Staubli VAL3: RemoteControl.pjx

--- RemoteControl.pjx ---
Parameters version=s8.10.3Cs9_BS2093 stackSize=5000 millimeterUnit=true
Program file=decodeBlend.pgx
Program file=decodeConfig.pgx
Program file=decodeDesc.pgx
Program file=decodeLocation.pgx
Program file=decodePose.pgx
Program file=decodeTool.pgx
Program file=encodeJoint.pgx
Program file=encodePoint.pgx
Program file=init.pgx
Program file=motionReporter.pgx
Program file=motionSupervisor.pgx
Program file=motionWorker.pgx
Program file=movingReporter.pgx
Program file=sendAck.pgx
Program file=sendError.pgx
Program file=sendMoving.pgx
Program file=sendPowerOff.pgx
Program file=sendStatus.pgx
Program file=socketHandler.pgx
Program file=start.pgx
Program file=stop.pgx
Data file=RemoteControl.dtx

--- RemoteControl.dtx ---
num VERSION = 1
sio socket = {link=UdpSocket\RemoteControl}
pointRx BASE_POSITION = {x=50, y=50, z=300, shoulder=sfree, elbow=efree, wrist=wfree, fatherId=world[0]}
jointRx BASE_POSE = {j1=-4.75879959898819E-06, j2=-86.5939224981684, j3=136.317941524159, j4=3.68060849006858E-06, j5=40.2759589805294, j6=-2.91771227743379E-06}
num MAGIC_HEADER = 149
string TASK_NAMES{}
  [MotionWorker] = "motionWorker"
  [MotionReporter] = "motionReporter"
  [MotionSupervisor] = "motionSupervisor"
  [SocketHandler] = "socketHandler"
  [MovingReporter] = "movingReporter"
tool endEffector = {x=660, fatherId=mount[0]}
tool mount = {ry=-90, fatherId=flange[0]}
bool motionQueued
num motionType
num reportInterval
pointRx target = {shoulder=sfree, elbow=efree, wrist=wfree, fatherId=world[0]}
mdesc NOMINAL_CONFIG = {accel=25, decel=25, blend=off}
mdesc SLOW_CONFIG = {accel=25, decel=25, tmax=150, rmax=50, blend=off}
mdesc moveConfig = {blend=off}
jointRx pose
tool selectedTool = {fatherId=flange[0]}
bool reportEnabled
configRx ARM_CONFIG = {shoulder=sfree, elbow=efree, wrist=wfree}
pointRx intermediate = {fatherId=world[0]}

--- start.pgx ---
program start()
begin
  logMsg("RemoteControl - Version " + toString("", VERSION))

  call init()
  enablePower()

  // Move to the initial starting pose
  logMsg("[INIT] Moving dangerously to starting position")
  movej(BASE_POSE, mount, SLOW_CONFIG)
  waitEndMove()

  taskCreate TASK_NAMES["SocketHandler"], 5, socketHandler()
  taskCreate TASK_NAMES["MotionWorker"], 10, motionWorker()
  taskCreate TASK_NAMES["MotionSupervisor"], 20, motionSupervisor()
  taskCreate TASK_NAMES["MovingReporter"], 29, movingReporter()
  taskCreate TASK_NAMES["MotionReporter"], 30, motionReporter()
end

--- decodeBlend.pgx ---
program decodeBlend(mdesc& value, num& buffer[])
  local num decodeBuffer[2]
begin
  if buffer[0] == 0
    value.blend = off
  elseIf buffer[0] == 1
    value.blend = joint
  elseIf buffer[0] == 2
    value.blend = Cartesian
  endIf

  fromBinary(buffer[1], 8, "4.0b", decodeBuffer)

  value.leave = decodeBuffer[0]
  value.reach = decodeBuffer[1]

  logMsg("B: (" + toString("", value.blend) + ", " + toString("", value.leave) + ", " + toString("", value.reach) + ")")
end

--- decodeConfig.pgx ---
program decodeConfig(pointRx& value, num& buffer[])
begin
  if buffer[0] == 0
    value.config.shoulder = sfree
  elseIf buffer[0] == 1
    value.config.shoulder = ssame
  elseIf buffer[0] == 2
    value.config.shoulder = righty
  elseIf buffer[0] == 3
    value.config.shoulder = lefty
  endIf

  if buffer[1] == 0
    value.config.elbow = efree
  elseIf buffer[1] == 1
    value.config.elbow = esame
  elseIf buffer[1] == 2
    value.config.elbow = epositive
  elseIf buffer[1] == 3
    value.config.elbow = enegative
  endIf

  if buffer[2] == 0
    value.config.wrist = wfree
  elseIf buffer[2] == 1
    value.config.wrist = wsame
  elseIf buffer[2] == 2
    value.config.wrist = wpositive
  elseIf buffer[2] == 3
    value.config.wrist = wnegative
  endIf

  logMsg("S: " + toString("", buffer[0]) + "  E: " + toString("", buffer[1]) + "  W: " + toString("", buffer[2]))
end

--- decodeDesc.pgx ---
program decodeDesc(mdesc& value, num& buffer[])
  local num decodeBuffer[3]
begin
  fromBinary(buffer, 8, "4.0b", decodeBuffer)

  value.tvel = decodeBuffer[0]
  value.rvel = decodeBuffer[1]

  fromBinary(buffer[8], 3, "1", decodeBuffer)
  value.accel = decodeBuffer[0]
  value.vel   = decodeBuffer[1]
  value.decel = decodeBuffer[2]

  logMsg("D: (" + toString("3", value.tvel) + ", " + toString("3", value.rvel) + ", " + toString("3", value.accel) + ", " + toString("3", value.vel) + ", " + toString("3", value.decel) + ")")
end

--- decodeLocation.pgx ---
program decodeLocation(point& value, num& buffer[])
  local num decodeBuffer[6]
begin
  fromBinary(buffer, 24, "4.0b", decodeBuffer)

  value.trsf = {decodeBuffer[0], decodeBuffer[1], decodeBuffer[2], decodeBuffer[3], decodeBuffer[4], decodeBuffer[5]}

  logMsg("P: (" + toString("3", value.trsf.x) + ", " + toString("3", value.trsf.y) + ", " + toString("3", value.trsf.z) + ")  R: (" + toString("3", value.trsf.rx) + ", " + toString("3", value.trsf.ry) + ", " + toString("3", value.trsf.rz) + ")")
end

--- decodePose.pgx ---
program decodePose(joint& value, num& buffer[])
  local num decodeBuffer[6]
begin
  fromBinary(buffer, 24, "4.0b", decodeBuffer)

  value = {decodeBuffer[0], decodeBuffer[1], decodeBuffer[2], decodeBuffer[3], decodeBuffer[4], decodeBuffer[5]}

  logMsg("J: (" + toString("3", value.j1) + ", " + toString("3", value.j2) + ", " + toString("3", value.j3) + ", " + toString("3", value.j4) + ", " + toString("3", value.j5) + ", " + toString("3", value.j6) + ")")
end

--- decodeTool.pgx ---
program decodeTool(tool& value, num& buffer[])
  local num decodeBuffer[6]
begin
  fromBinary(buffer, 24, "4.0b", decodeBuffer)

  value.trsf = {decodeBuffer[0], decodeBuffer[1], decodeBuffer[2], decodeBuffer[3], decodeBuffer[4], decodeBuffer[5]}

  logMsg("P: (" + toString("3", value.trsf.x) + ", " + toString("3", value.trsf.y) + ", " + toString("3", value.trsf.z) + ")  R: (" + toString("3", value.trsf.rx) + ", " + toString("3", value.trsf.ry) + ", " + toString("3", value.trsf.rz) + ")")
end

--- encodeJoint.pgx ---
program encodeJoint(joint& value, num& buffer[])
  local num elements[6]
begin
  elements[0] = value.j1
  elements[1] = value.j2
  elements[2] = value.j3
  elements[3] = value.j4
  elements[4] = value.j5
  elements[5] = value.j6

  toBinary(elements, 6, "4.0b", buffer)
end

--- encodePoint.pgx ---
program encodePoint(point& value, num& buffer[])
  local num elements[6]
begin
  elements[0] = value.trsf.x
  elements[1] = value.trsf.y
  elements[2] = value.trsf.z
  elements[3] = value.trsf.rx
  elements[4] = value.trsf.ry
  elements[5] = value.trsf.rz

  toBinary(elements, 6, "4.0b", buffer)
end

--- init.pgx ---
program init()
begin
  moveConfig = NOMINAL_CONFIG
  motionQueued = false
  reportEnabled = false
  reportInterval = 0.1
  selectedTool = endEffector
  target.config = ARM_CONFIG
end

--- motionReporter.pgx ---
program motionReporter()
begin
  while true
    wait(reportEnabled)

    while reportEnabled
      call sendStatus()
      delay(reportInterval)
    endWhile
  endWhile
end

--- motionSupervisor.pgx ---
program motionSupervisor()
  local num buffer[8]
  local num value
begin
  while true
    // Sleep until the task enters a runtime error state
    wait(taskStatus(TASK_NAMES["MotionWorker"]) > 1)

    // Clear any invalid pending trajectories
    resetMotion()

    // Notify any clients of the error
    call sendError(1, taskStatus(TASK_NAMES["MotionWorker"]))

    // Resume the task from the next line
    taskResume(TASK_NAMES["MotionWorker"], 1)
  endWhile
end

--- motionWorker.pgx ---
program motionWorker()
begin

  while true
    wait(motionQueued)
    motionQueued = false

    if motionType == 0
      logMsg("[MOTION] Linear move")
      movel(target, selectedTool, moveConfig)

    elseIf motionType == 1
      logMsg("[MOTION] Direct move")
      movej(target, selectedTool, moveConfig)

    elseIf motionType == 2
      logMsg("[MOTION] Joint move")
      movej(pose, selectedTool, moveConfig)

    elseIf motionType == 3
      logMsg("[MOTION] Circular move")
      movec(intermediate, target, selectedTool, moveConfig)
    endIf

  endWhile
end

--- movingReporter.pgx ---
program movingReporter()
  local bool settled
begin
  settled = false

  while true
    wait(isSettled() != settled)
    settled = !settled

    call sendMoving()
  endWhile
end

--- sendAck.pgx ---
program sendAck(num id)
  local num buffer[3]
begin
  buffer[0] = MAGIC_HEADER
  buffer[1] = 128
  buffer[2] = id
  sioSet(socket, buffer)
end

--- sendComplete.pgx ---
program sendComplete()
  local num buffer[2]
begin
  buffer[0] = MAGIC_HEADER
  buffer[1] = 2
  sioSet(socket, buffer)
end

--- sendError.pgx ---
program sendError(num code, num argument)
  local num buffer[5]
begin
  buffer[0] = MAGIC_HEADER
  buffer[1] = 129
  buffer[2] = code

  toBinary(argument, 1, "2b", buffer[3])

  sioSet(socket, buffer)
end

--- sendMoving.pgx ---
program sendMoving()
  local num buffer[4]
begin
  buffer[0] = MAGIC_HEADER
  buffer[1] = 132
  buffer[2] = sel(isSettled(), 1, 0)
  sioSet(socket, buffer)
end

--- sendPowerOff.pgx ---
program sendPowerOff()
  local num buffer[2]
begin
  buffer[0] = MAGIC_HEADER
  buffer[1] = 130
  sioSet(socket, buffer)
end

--- sendStatus.pgx ---
program sendStatus()
  local num buffer[79]
  local point currentPosition
  local joint currentPose
  local num moveId
begin
  buffer[0] = MAGIC_HEADER
  buffer[1] = 131

  currentPosition = here(endEffector, world)
  call encodePoint(currentPosition, buffer[2])

  currentPose = herej()
  call encodeJoint(currentPose, buffer[26])

  currentPose = getPositionErr()
  call encodeJoint(currentPose, buffer[50])

  buffer[74] = sel(isSettled(), 1, 0)

  moveId = getMoveId()
  toBinary(moveId, 1, "4.0b", buffer[75])

  sioSet(socket, buffer)
end

--- socketHandler.pgx ---
program socketHandler()
  local bool ack
  local num buffer[1024]
  local num bytesRead
  local num payloadSize
begin
  while true
    ack = true
    bytesRead = sioGet(socket, buffer)

    if bytesRead > 0
      logMsg("[SOCKET] UDP packet (" + toString("", bytesRead) + " B)")
    endIf

    if bytesRead >= 3
      payloadSize = bytesRead - 3
    endIf

    if bytesRead < 3
      logMsg("[SOCKET] Too few bytes read, misconfigured socket timeout?", 2)
      ack = false

    elseIf buffer[0] != MAGIC_HEADER
      logMsg("[SOCKET] Missing magic header", 3)
      ack = false

    elseIf buffer[2] == 0 and payloadSize == 0
      logMsg("[SOCKET] Handshake request")

    elseIf buffer[2] == 1 and payloadSize == 1
      logMsg("[SOCKET] Halt request")

      if buffer[3] == 1
        logMsg("[STOP] Returning to start")
        call sendAck(buffer[1])
        resetMotion()
        enablePower()
        movej(BASE_POSE, mount, SLOW_CONFIG)
        waitEndMove()
      endIf

      // Manually create the program stop task
      taskCreate "~RemoteControl", 1, stop()
      return

    elseIf buffer[2] == 2 and payloadSize == 1
      logMsg("[SOCKET] Move home request")

      wait(!motionQueued)

      motionType = buffer[3]
      moveConfig.blend = off

      if motionType == 2
        pose = BASE_POSE
      else
        target = BASE_POSITION
      endIf

      selectedTool = mount
      motionQueued = true

    elseIf buffer[2] == 3 and payloadSize == 1
      logMsg("[SOCKET] Set reporting request")
      reportEnabled = buffer[3] != 0

    elseIf buffer[2] == 4 and payloadSize == 4
      logMsg("[SOCKET] Set report frequency request")
      fromBinary(buffer[3], 4, "4.0b", reportInterval)

    elseIf buffer[2] == 5 and payloadSize == 3
      logMsg("[SOCKET] Configuration request")
      call decodeConfig(target, buffer[3])

    elseIf buffer[2] == 6 and payloadSize == 11
      logMsg("[SOCKET] Set profile")
      call decodeDesc(moveConfig, buffer[3])

    elseIf buffer[2] == 7 and payloadSize == 9
      logMsg("[SOCKET] Blending request")
      call decodeBlend(moveConfig, buffer[3])

    elseIf buffer[2] == 8 and payloadSize == 24
      logMsg("[SOCKET] Tool offset request")
      call decodeTool(endEffector, buffer[3])


    elseIf buffer[2] == 32 and payloadSize == 24
      logMsg("[SOCKET] Direct move request")

      wait(!motionQueued)
      call decodeLocation(target, buffer[3])

      motionType = 1
      selectedTool = endEffector
      motionQueued = true

    elseIf buffer[2] == 33 and payloadSize == 24
      logMsg("[SOCKET] Linear move request")

      wait(!motionQueued)
      call decodeLocation(target, buffer[3])

      motionType = 0
      selectedTool = endEffector
      motionQueued = true

    elseIf buffer[2] == 34 and payloadSize == 24
      logMsg("[SOCKET] Joint move request")

      wait(!motionQueued)
      call decodePose(pose, buffer[3])

      motionType = 2
      selectedTool = endEffector
      motionQueued = true

    elseIf buffer[2] == 35 and payloadSize == 48
      logMsg("[SOCKET] Circular movement request")

      wait(!motionQueued)

      call decodeLocation(intermediate, buffer[3])
      call decodeLocation(target, buffer[27])

      motionType = 3
      selectedTool = endEffector
      motionQueued = true


    else
      logMsg("[SOCKET] Unknown message: " + toString("", buffer[2]) + " with payload size " + toString("", payloadSize), 3)
      ack = false

    endIf

    if ack
      call sendAck(buffer[1])
    endIf

  endWhile
end

--- stop.pgx ---
program stop()
  local string key
begin
  key = first(TASK_NAMES)

  while key != ""
    taskKill(TASK_NAMES[key])
    key = next(TASK_NAMES[key])
  endWhile

  disablePower()

  // call sendPowerOff()
end
